Staubli VAL3: toPointRxEuler.pgx

public program toPointRxEuler(num& x_nQuaternion[], pointRx& x_pPointRx)
  local num l_nT0
  local num l_nT1
  local num l_nT2
  local num l_nT3
  local num l_nT4
  local num l_nAtan2Res
  local num _EPS
  local num si
  local num sj
  local num sk
  local num ci
  local num cj
  local num ck
  local num M02
  local num M12
  local num M22
  local num cy
  local num ax
  local num ay
  local num az
begin
  _EPS = 1e-16

  l_nT0 = 2 * (x_nQuaternion[3] * x_nQuaternion[0] + x_nQuaternion[1] * x_nQuaternion[2])
  l_nT1 = 1 - 2 * (x_nQuaternion[0] * x_nQuaternion[0] + x_nQuaternion[1] * x_nQuaternion[1])
  call atan2(l_nT0, l_nT1, l_nAtan2Res)
  si = sin(l_nAtan2Res)
  ci = cos(l_nAtan2Res)

  l_nT2 = 2 * (x_nQuaternion[3] * x_nQuaternion[1] - x_nQuaternion[2] * x_nQuaternion[0])
  sj = limit(l_nT2, -1, 1)
  cj = cos(asin(sj))

  l_nT3 = 2 * (x_nQuaternion[3] * x_nQuaternion[2] + x_nQuaternion[0] * x_nQuaternion[1])
  l_nT4 = 1 - 2 * (x_nQuaternion[1] * x_nQuaternion[1] + x_nQuaternion[2] * x_nQuaternion[2])
  call atan2(l_nT3, l_nT4, l_nAtan2Res)
  sk = sin(l_nAtan2Res)
  ck = cos(l_nAtan2Res)

  // extrinsic2intrinsic
  M02 = sj * ci * ck + si * sk
  M12 = sj * ci * sk - si * ck
  M22 = cj * ci

  cy = sqrt(M22 * M22 + M12 * M12)

  if cy > _EPS
    call atan2(M12, M22, ax)
    call atan2(-M02, cy, ay)
    call atan2(sj * (si * ck) - (ci * sk), cj * ck, az)
  else
    ax = 0.0
    call atan2(-M02, cy, ay)
    call atan2(-cj * sk, sj * si * sk + ci * ck, az)
  endIf

  x_pPointRx.trsf.rx = ax * -1
  x_pPointRx.trsf.ry = ay * -1
  x_pPointRx.trsf.rz = az * -1

end
